FUNCTION_BLOCK {BlockName} (* {Description} *)
  (* Standard: 61499-2 *)
  (* Version 0.0, {MM/DD/YYYY}, {Author}, {YourOrg}, Initial version *)
  PACKAGE {YourNamespace};
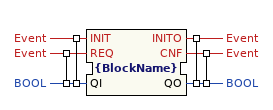
  EVENT_INPUT
    INIT WITH QI; (* Initialization Request *)
    REQ WITH QI; (* Normal Execution Request *)
  END_EVENT
  EVENT_OUTPUT
    INITO WITH QO; (* Initialization Confirm *)
    CNF WITH QO; (* Execution Confirmation *)
  END_EVENT
  VAR_INPUT
    QI : BOOL; (* Input event qualifier *)
  END_VAR
  VAR_OUTPUT
    QO : BOOL; (* Output event qualifier *)
  END_VAR
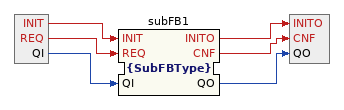
  FBS
    subFB1 : {SubFBType};
  END_FBS
  EVENT_CONNECTIONS
    INIT TO subFB1.INIT;
    REQ TO subFB1.REQ;
    subFB1.INITO TO INITO;
    subFB1.CNF TO CNF;
  END_CONNECTIONS
  DATA_CONNECTIONS
    QI TO subFB1.QI;
    subFB1.QO TO QO;
  END_CONNECTIONS
END_FUNCTION_BLOCK
(* other elements stored in the file *)
(* Layout Conventions: - Inputs:  x=100, events y=200+100*i, data y=500+100*i - FBs:     x=500+400*i, y=350 - Outputs: x=800 (1 FB) or 500+(fbCount-1)*400+400, events y=200+100*i, data y=500+100*i *)
(* FB instances: x = 500 + (index * 400), y = 350 *)
(* Input events: x=100, y = 200 + (index * 100) *)
(* Input data: x=100, y = 500 + (index * 100) *)
(* Output events: x=800 (for 1 FB), y = 200 + (index * 100) *)
(* Output data: x=800 (for 1 FB), y = 500 + (index * 100) *)
